FUNCTION_BLOCK FB_FileHandle
VAR
	_sNetID: T_AmsNetId;
	_ErrorMessage: STRING;
	_bError: BOOL;
	_bFileOpened: BOOL;
	_bFileClosed: BOOL;
	_sWrite: STRING;
	_bDirectoryCreated: BOOL;
	sFileName: STRING;
	sDirectory: STRING;
	hFile: UINT;
	fbCreateDirectory: FB_CreateDir;
	fbFileOpen: FB_FileOpen;
	fbFileWrite: FB_FileWrite;
	fbFileClose: FB_FileClose;
END_VAR

METHOD FB_init : BOOL
VAR_INPUT
	/// if TRUE, the retain variables are initialized (warm start / cold start)
	bInitRetains: BOOL;
	/// if TRUE, the instance afterwards gets moved into the copy code (online change)
	bInCopyCode: BOOL;
	Directory: STRING;
	FileName: STRING;
END_VAR
M_SetPath(Directory, FileName);
END_METHOD

PROPERTY isErrorOccured : BOOL
GET
isErrorOccured := This^._bError;
END_GET
END_PROPERTY

PROPERTY isFileClosed : BOOL
GET
isFileClosed := This^._bFileClosed;
END_GET
END_PROPERTY

PROPERTY isFileOpened : BOOL
GET
isFileOpened := This^._bFileOpened;
END_GET
END_PROPERTY

METHOD M_FileClose
fbFileClose(
	sNetId:= _sNetId, 
	hFile:= hFile, 
	bExecute:= TRUE, 
	tTimeout:= , 
	bBusy=> , 
	bError=> , 
	nErrId=> );
	
IF fbFileClose.bError THEN
	_ErrorMessage := CONCAT('FileOpen Failed ErrID = ', UDINT_TO_STRING(fbFileClose.nErrId));
	_bError := TRUE;
	fbFileClose(bExecute := FALSE);
	Return;
END_IF

IF fbFileClose.bBusy THEN
	RETURN;
ELSE
	_bFileClosed := TRUE;
	_bFileOpened := FALSE;
END_IF
END_METHOD

METHOD M_FileOpen
IF NOT _bDirectoryCreated THEN
	fbCreateDirectory(sPathName := THIS^.sDirectory ,bExecute := TRUE);
	
	IF fbCreateDirectory.bBusy THEN
		_bDirectoryCreated := FALSE;
		RETURN;	
	ELSE 
		fbCreateDirectory(bExecute := FALSE);
		_bDirectoryCreated := TRUE;
	END_IF
ELSE
	fbFileOpen(
		sNetId:= , 
		sPathName:= P_FilePath, 
		nMode:= FOPEN_MODEAPPEND OR FOPEN_MODETEXT , 
		ePath:=PATH_GENERIC, 
		bExecute:= TRUE, 
		tTimeout:= , 
		bBusy=> , 
		bError=> , 
		nErrId=> , 
		hFile=> hFile);
	
	IF fbFileOpen.bError THEN
		_ErrorMessage := CONCAT('FileOpen Failed ErrID = ', UDINT_TO_STRING(fbFileOpen.nErrId));
		RETURN;
	END_IF
		
	IF fbFileOpen.bBusy THEN
		RETURN;
	ELSE
		fbFileOpen(bExecute := FALSE);
		_bFileOpened := TRUE;
		_bFileClosed := FALSE;
	END_IF
END_IF
END_METHOD

METHOD M_FileWrite
IF _sWrite <> '' THEN
	fbFileWrite(
		sNetId:= _sNetID, 
		hFile:= hFile, 
		pWriteBuff:= ADR(_sWrite) , 
		cbWriteLen:= INT_TO_UDINT(LEN(_sWrite)), 
		bExecute:= TRUE, 
		tTimeout:= , 
		bBusy=> , 
		bError=> , 
		nErrId=> , 
		cbWrite=> );
		
	IF fbFileWrite.bError THEN
		_ErrorMessage := CONCAT('FileWrite Failed ErrID = ', UDINT_TO_STRING(fbFileWrite.nErrId));
		Return;
	END_IF
	
	IF fbFileWrite.bBusy THEN
		RETURN;
	ELSE
		fbFileWrite(bExecute := FALSE);
		_sWrite := '';  //Reset sWrite after file write
	END_IF
END_IF
END_METHOD

METHOD PRIVATE M_SetPath
VAR_INPUT
	sDirectory: STRING;
	sFileName: STRING;
END_VAR
THIS^.sDirectory := sDirectory;
THIS^.sFileName := sFileName;
END_METHOD

PROPERTY P_ErrorMessage : T_Maxstring
GET
P_ErrorMessage := _ErrorMessage;
END_GET
END_PROPERTY

PROPERTY P_FilePath : STRING
GET
P_FilePath := CONCAT(This^.sDirectory, CONCAT('/', This^.sFileName));
END_GET
END_PROPERTY

PROPERTY P_sNetID : T_AmsNetID
GET
P_sNetID := This^._sNetID;
END_GET
SET
 This^._sNetID :=P_sNetID;
END_SET
END_PROPERTY

PROPERTY P_SomethingToWrite : T_Maxstring
GET
P_SomethingToWrite:= This^._sWrite ;
END_GET
SET
This^._sWrite := P_SomethingToWrite;
END_SET
END_PROPERTY

END_FUNCTION_BLOCK

(* stored: Version 1.1.0.1, ProductVersion 3.1.4024.12
   POU FB_FileHandle: Id {6e354855-d896-4c11-9eb6-3c21cbff619a}, SpecialFunc None
   Method FB_init: Id {9b9fadf7-825a-48d7-b801-6328987d722b}
   Property isErrorOccured: Id {cdcc4e3e-e26b-49ea-b6f9-b8d42764b31c}
   Get Get: Id {bc410799-e964-4627-8878-7cde17a17db4}
   Property isFileClosed: Id {bce0b5a9-9157-4340-b16b-e365091fabf4}
   Get Get: Id {fedacfe5-9b34-445b-b0de-d4f2661137b7}
   Property isFileOpened: Id {56fe483f-c565-4b1b-84e9-a4835f9a4735}
   Get Get: Id {c2f8d079-8224-4ee9-ac2d-d5d39ffad1e4}
   Method M_FileClose: Id {5d157b2a-2771-4a2c-bc30-1c8d0c9b1edc}
   Method M_FileOpen: Id {74f81313-f49f-471d-b6bc-904b3e857261}
   Method M_FileWrite: Id {35b963a3-f675-4192-9c21-765ba48c8f7a}
   Method M_SetPath: Id {6170592f-9344-4294-bdef-e818e6334847}
   Property P_ErrorMessage: Id {2d708a9a-fe87-433f-a267-8a592eeb1175}
   Get Get: Id {cb38d3e2-c7c8-4bdd-a40d-e9735a400745}
   Property P_FilePath: Id {cb7e9d2b-4c47-4dcb-8623-7a8e8d4a92fe}
   Get Get: Id {d86e9153-5077-43bc-8ac1-9185743e5b31}
   Property P_sNetID: Id {20b7f168-63ae-4c81-8c01-791f2a11491b}
   Get Get: Id {f900ce5e-d8c7-49f0-a8c4-08c647404a7b}
   Set Set: Id {4b90a82e-ec70-4c3f-be59-8271d2b76c0b}
   Property P_SomethingToWrite: Id {ff3f8e55-63cc-4185-b7a2-2bd159723e90}
   Get Get: Id {3f8eb8ae-b2b1-4edf-ae60-7b51551fa729}
   Set Set: Id {819b5759-4e6c-4555-99b5-a880ab01217b} *)
